//---------------------------------------------------------------------------------------------------------------
//
//  HAUD 2026.04.10.
//
//  fb_XmlBase
//    - wraps xml read
//    - wraps xml write
//
//   - abstract base class for extending xml R/W ctrl for any data
//
//---------------------------------------------------------------------------------------------------------------
// This SOFTWARE is provided as an Example by THE PROVIDER "as is" and "with all faults." THE PROVIDER makes no 
// representations or warranties of any kind concerning the safety, suitability, lack of viruses, inaccuracies, 
// typographical errors, or other harmful components of this SOFTWARE. There are inherent dangers in the use of 
// any software, and you are solely responsible for determining whether this SOFTWARE is compatible with your 
// equipment and other software installed on your equipment. You are also solely responsible for the protection 
// of your equipment and backup of your data, and THE PROVIDER will not be liable for any damages you may suffer 
// in connection with using, modifying, or distributing this SOFTWARE.
//---------------------------------------------------------------------------------------------------------------
FUNCTION_BLOCK ABSTRACT fb_XmlBase
VAR
  //------------------------------------------------------------------------------------------------------------
  // pointer check result
  //------------------------------------------------------------------------------------------------------------
  _eCheck                     : E_DATA_CHECK;
  _sCheck                     : STRING;
  //------------------------------------------------------------------------------------------------------------
  // internal control and state
  //------------------------------------------------------------------------------------------------------------
  _eInit                      : E_PROGRESS;
  _eCmd,
  _eCmdOld                    : E_DATA_CTRL;
  _eState                     : E_DATA_STATE;
  _eResult                    : E_PROGRESS;
  //------------------------------------------------------------------------------------------------------------
  // Tc2_XmlDataSrv wrappers
  //------------------------------------------------------------------------------------------------------------
  _fbXmlRead                  : fb_XmlRead;
  _fbXmlWrite                 : fb_XmlWrite;
  //------------------------------------------------------------------------------------------------------------
  // who am I?
  //  - Identity built in extending class
  //
  // see fb_Configuration.Identity.Set() as example
  //------------------------------------------------------------------------------------------------------------
  {attribute 'displaymode' := 'hex'}
  _XpuIdentity                : OTCID;        // identity must be set by extending class
  _sIdentity                  : STRING;       // part of filename
  //------------------------------------------------------------------------------------------------------------
  // where am I?
  //  - hocus pocus
  //    - you have to define my locus 
  //
  // see fb_Configuration.Identity.Set() as example
  //------------------------------------------------------------------------------------------------------------
  _sDirectoryPath             : STRING;       // root directory for data
  _sFilePath                  : STRING(255);  // path and filename (shall include identity in filepath)

  _sName                      : STRING;       // filename with *.xml
  _sXpath                     : STRING;       // XPath from extending class
  //------------------------------------------------------------------------------------------------------------
  // what am I?
  //  - data from the void
  //------------------------------------------------------------------------------------------------------------
  _pData                      : Global.PVOID;
  _nData                      : UDINT;
  //------------------------------------------------------------------------------------------------------------
  _eDeviceIdentifier          : e_Device;
  _stMsg                      : ST_Message;
  _eMessageLevel              : E_MessageType;
END_VAR

METHOD CreateFolder : E_PROGRESS
VAR_INPUT
  Execute         : BOOL;
END_VAR
VAR_INST
  _nErrorId       : UDINT;
  _eState         : E_PROGRESS;
  _sPath          : Tc2_System.T_MaxString;
  _fbCreateDir    : Tc2_System.FB_CreateDir;
END_VAR

IF NOT Execute
THEN
  _eState                     := E_PROGRESS.PROGRESS_INIT;
END_IF


CASE _eState
OF
  E_PROGRESS.PROGRESS_INIT:
    IF Execute
    THEN
      _eState                 := E_PROGRESS.PROGRESS_BUSY;
      _nErrorId               := 0;

      _fbCreateDir(
                    sNetId    := '', 
                    sPathName := _sPath, 
                    ePath     := Tc2_System.E_OpenPath.PATH_GENERIC, 
                    bExecute  := FALSE, 
                    tTimeout  := T#1S);
    END_IF

  E_PROGRESS.PROGRESS_BUSY:
    _fbCreateDir(
                  sNetId      := '', 
                  sPathName   := _sPath, 
                  ePath       := Tc2_System.E_OpenPath.PATH_GENERIC, 
                  bExecute    := TRUE, 
                  tTimeout    := T#1S,
                  nErrId      => _nErrorId);

    IF _fbCreateDir.bBusy
    THEN
      _eState                 := E_PROGRESS.PROGRESS_OCCUPIED;
    END_IF

  E_PROGRESS.PROGRESS_OCCUPIED:
    _fbCreateDir(
                  sNetId      := '', 
                  sPathName   := _sPath, 
                  ePath       := Tc2_System.E_OpenPath.PATH_GENERIC, 
                  bExecute    := TRUE, 
                  tTimeout    := T#1S,
                  nErrId      => _nErrorId);

    IF NOT _fbCreateDir.bBusy
    THEN
      _eState                 := E_PROGRESS.PROGRESS_WORKING;
    END_IF

  E_PROGRESS.PROGRESS_WORKING:
    _eState                   := E_PROGRESS.PROGRESS_DONE;
    _fbCreateDir(
                  sNetId      := '', 
                  sPathName   := _sPath, 
                  ePath       := Tc2_System.E_OpenPath.PATH_GENERIC, 
                  bExecute    := FALSE, 
                  tTimeout    := T#1S);

    IF (_eMessageLevel > E_MessageType.eMessageError)
    THEN
      _stMsg.eType            := E_MessageType.eMessageInfo;
      _stMsg.eDevice          := _eDeviceIdentifier;
      _stMsg.eSubdevice       := e_Subdevice.fbCreateFolder;
      _stMsg.iErrorNumber     := 0;
      _stMsg.sText            := concat(' : ', TO_STRING(_eState));
      f_MessageSet(_stMsg);
    END_IF
END_CASE

CreateFolder                  := _eState;
END_METHOD

PROPERTY FilePath : string(255)
GET
FilePath := _sFilePath;
END_GET
END_PROPERTY

PROPERTY FolderPath : string
GET
FolderPath := _sDirectoryPath;
END_GET
SET
_sDirectoryPath := FolderPath;
END_SET
END_PROPERTY

PROPERTY MessageDevice : udint
SET
_eDeviceIdentifier   := MessageDevice;
END_SET
END_PROPERTY

PROPERTY MessageLevel : e_messagetype
SET
_eMessageLevel := MessageLevel;
END_SET
END_PROPERTY

METHOD XmlRead  : E_PROGRESS
VAR_INPUT
  Execute               : BOOL;
END_VAR
VAR_INST
  _eState               : E_PROGRESS;
  _nErrorId             : UDINT;
END_VAR

IF NOT Execute
THEN
  _eState                     := E_PROGRESS.PROGRESS_INIT;
END_IF

CASE _eState
OF
  E_PROGRESS.PROGRESS_INIT:
    IF Execute
    THEN
      _nErrorId               := 0;
      _eState                 := E_PROGRESS.PROGRESS_BUSY;

      IF (_eMessageLevel > E_MessageType.eMessageInfo)
      THEN
        _stMsg.eType          := E_MessageType.eMessageVerbose;
        _stMsg.eDevice        := _eDeviceIdentifier;
        _stMsg.eSubdevice     := e_Subdevice.fbXmlRead;
        _stMsg.iErrorNumber   := _nErrorId;
        _stMsg.sText          := concat(' : ', TO_STRING(_eState));
        f_MessageSet(_stMsg);
      END_IF
    END_IF

  E_PROGRESS.PROGRESS_BUSY:
    _eState                   := E_PROGRESS.PROGRESS_OCCUPIED;
    _fbXmlRead(
              bExecute        := FALSE, 
              sFilePath       := _sFilePath, 
              sXPath          := _sXpath, 
              pData           := _pData, 
              diSize          := _nData);

  E_PROGRESS.PROGRESS_OCCUPIED:
    _fbXmlRead(
              bExecute        := TRUE);

    IF _fbXmlRead.bError
    THEN
      _nErrorId               := _fbXmlRead.nError;
      _eState                 := E_PROGRESS.PROGRESS_ERROR;

      _stMsg.eType            := E_MessageType.eMessageError;
      _stMsg.eDevice          := _eDeviceIdentifier;
      _stMsg.eSubdevice       := e_Subdevice.fbXmlRead;
      _stMsg.iErrorNumber     := _nErrorId;
      _stMsg.sText            := concat(' : ', TO_STRING(_eState));
      f_MessageSet(_stMsg);

      _fbXmlRead(
              bExecute        := FALSE);

    ELSIF _fbXmlRead.bDone
    THEN
      _eState                 := E_PROGRESS.PROGRESS_WORKING;
      _fbXmlRead(
              bExecute        := FALSE);
    END_IF

  E_PROGRESS.PROGRESS_WORKING:
    _eState                   := E_PROGRESS.PROGRESS_DONE;

    IF (_eMessageLevel > E_MessageType.eMessageError)
    THEN
      _stMsg.eType            := E_MessageType.eMessageInfo;
      _stMsg.eDevice          := _eDeviceIdentifier;
      _stMsg.eSubdevice       := e_Subdevice.fbXmlRead;
      _stMsg.iErrorNumber     := _nErrorId;
      _stMsg.sText            := concat(' : ', TO_STRING(_eState));
      f_MessageSet(_stMsg);
    END_IF
END_CASE

XmlRead                       := _eState;
END_METHOD

METHOD XmlWrite : E_PROGRESS
VAR_INPUT
  Execute               : BOOL;
END_VAR
VAR_INST
  _eState               : E_PROGRESS;
  _nErrorId             : UDINT;
END_VAR

IF NOT Execute
THEN
  _eState                     := E_PROGRESS.PROGRESS_INIT;
END_IF

CASE _eState
OF
  E_PROGRESS.PROGRESS_INIT:
    IF Execute
    THEN
      _nErrorId               := 0;
      _eState                 := E_PROGRESS.PROGRESS_BUSY;

      IF (_eMessageLevel > E_MessageType.eMessageInfo)
      THEN
        _stMsg.eType          := E_MessageType.eMessageVerbose;
        _stMsg.eDevice        := _eDeviceIdentifier;
        _stMsg.eSubdevice     := e_Subdevice.fbXmlWrite;
        _stMsg.iErrorNumber   := _nErrorId;
        _stMsg.sText          := concat(' : ', TO_STRING(_eState));
        f_MessageSet(_stMsg);
      END_IF
    END_IF

  E_PROGRESS.PROGRESS_BUSY:
    _eState                   := E_PROGRESS.PROGRESS_OCCUPIED;
    _fbXmlWrite(
              bExecute        := FALSE, 
              sFilePath       := _sFilePath, 
              sXPath          := _sXpath, 
              pData           := _pData, 
              diSize          := _nData);

  E_PROGRESS.PROGRESS_OCCUPIED:
    _fbXmlWrite(
              bExecute        := TRUE);

    IF _fbXmlWrite.bError
    THEN
      _nErrorId               := _fbXmlRead.nError;
      _eState                 := E_PROGRESS.PROGRESS_ERROR;

      _stMsg.eType            := E_MessageType.eMessageError;
      _stMsg.eDevice          := _eDeviceIdentifier;
      _stMsg.eSubdevice       := e_Subdevice.fbXmlWrite;
      _stMsg.iErrorNumber     := _nErrorId;
      _stMsg.sText            := concat(' : ', TO_STRING(_eState));
      f_MessageSet(_stMsg);

      _fbXmlWrite(
              bExecute        := FALSE);

    ELSIF _fbXmlWrite.bDone
    THEN
      _eState                 := E_PROGRESS.PROGRESS_WORKING;
      _fbXmlWrite(
              bExecute        := FALSE);
    END_IF

  E_PROGRESS.PROGRESS_WORKING:
    _eState                   := E_PROGRESS.PROGRESS_DONE;

    IF (_eMessageLevel > E_MessageType.eMessageError)
    THEN
      _stMsg.eType            := E_MessageType.eMessageInfo;
      _stMsg.eDevice          := _eDeviceIdentifier;
      _stMsg.eSubdevice       := e_Subdevice.fbXmlWrite;
      _stMsg.iErrorNumber     := _nErrorId;
      _stMsg.sText            := concat(' : ', TO_STRING(_eState));
      f_MessageSet(_stMsg);
    END_IF
END_CASE

XmlWrite                      := _eState;
END_METHOD

END_FUNCTION_BLOCK

(* stored: Version 1.1.0.1
   POU fb_XmlBase: Id {a411dbad-6751-4f66-9ce6-10c9e989d98d}, SpecialFunc None
   Folder methods: Id {ddf31a72-4ff3-4f92-b12f-f19e5140afbf}
   Folder properties: Id {94e7d8b5-e77d-4565-b5ef-edd730b87e43}
   Method CreateFolder: Id {9336a9b9-a4f4-4ecd-8f18-2087cc7da1a8}
   Property FilePath: Id {43658111-e80d-4c31-8ff6-dcdf07371bb2}
   Get Get: Id {f398be6f-7cf8-4a1e-8a83-56f354118171}
   Property FolderPath: Id {e27c21b9-2599-4ab8-b4d7-8aae8580ded4}
   Get Get: Id {2dee3ff3-6f9a-46eb-8993-bd9fcbbbaf7b}
   Set Set: Id {c3670cba-402f-4be0-965a-134ec240135b}
   Property MessageDevice: Id {097bc27a-b3d1-4cc7-afa7-35376dec7a92}
   Set Set: Id {2a869d90-c5c5-49c4-a4f5-12d8df205078}
   Property MessageLevel: Id {66cbafc1-ae1c-4abc-baa4-7e5501ee8181}
   Set Set: Id {9cd0d71c-f3d7-483d-9245-759f67d862ea}
   Method XmlRead: Id {698228e2-8548-4e36-a36a-bcfac941d13d}
   Method XmlWrite: Id {9b2aef7b-591c-489a-8d94-197487238165} *)
